TYPE E_ITC_ElementControlCode :
(**************************************************************************************
 * 	Application		:	BoxControl Framework
 *	Revision		:	$Revision: 404529 $
 *	Revision date	:	$Date: 2018-04-23 08:21:38 +0200 (Mo., 23 Apr 2018) $
 *	Last changed by	:	$Author: b7bolm $
 *	URL				:	$URL: http://almscdc.swisslog.com/repo/SWPD/Development/BoxControlFramework/20_Release/trunk/01_Software/BCF/BCF/JumpStart/20_Product/10_App/13_Elements/10_Lib/10_Conv/01_DUTs/E_ITC_ElementControlCode.TcDUT $
 *
 *	Purpose			:	Element control code
 *
 * ------------------------------------------------------------------------------------
 *	Copyright Swisslog [IP AG], Switzerland. All rights reserved.
 * 
 * ------------------------------------------------------------------------------------
 *	
 * 	Revision History: 
 *
 * 	VERSION			DATE			INITIALS			DESCRIPTION
 *	0.1				01.01.2001		swl					Example
 *
 **************************************************************************************)
(
	NO_CODE					:= 0, // No code
	RESET_ERROR 			:= 1, // Acknowledge Error
	INITIALIZE				:= 2, // Initialize
	ENABLE					:= 4, // E.g. start, stop
	SET_VARIABLE			:= 5, // Set Variable
	SET_ERROR				:= 20 // Set error
);
END_TYPE

(* stored: Version 1.1.0.1, ProductVersion 3.1.4022.12
   DUT E_ITC_ElementControlCode: Id {a7d7d51a-90d6-432b-a10c-79de81b7d57e} *)
